FUNCTION_BLOCK TcoTixonVibro_v_1_x_x EXTENDS TcoCore.TcoComponent
VAR_INPUT
    inControllerInAuto : BOOL;
    inNotEmptyFeeder : BOOL;
    inSeparatorHomePos : BOOL;
    inFillingSensor : BOOL;
    inSeparatorPresent : BOOL;
    inComponentOutOfBox : BOOL;
    inSeparatorWorkPos : BOOL;
END_VAR
VAR_OUTPUT
    outFeedingA : BOOL;
    outSepareComponent : BOOL;
    outBlowValveA : BOOL;
    outRedLed : BOOL;
    outGreenLed : BOOL;
    outHopper : BOOL;
    outShotComponent : BOOL;
END_VAR
VAR
    {attribute addProperty Name "<#Status#>"}
    {attribute clr [ReadOnly()]}
    _status : TcoTixonVibro_Status_v_1_x_x;
    {attribute addProperty Name "<#Control#>"}
    _control : TcoTixonVibro_Control_v_1_x_x;
    {attribute addProperty Name "<#Config#>"}
    _config : TcoTixonVibro_Config_v_1_x_x;
    _someTaskIsActive : BOOL;
    {attribute 'hide'}
    _blink : TcoUtilities.TcoBlinker(THIS^);
    _runAutomatic : BOOL;
    _hasError : BOOL;
END_VAR
VAR
    {attribute addProperty Name "<#Separator task#>"}
    _separatorTask : TcoTixonVibroSeparatorTask(THIS^);
    {attribute addProperty Name "<#Buffer task#>"}
    _bufferTask : TcoTixonBufferTask(THIS^);
    {attribute addProperty Name "<#Hopper task#>"}
    _hopperTask : TcoTixonHopperTask(THIS^);
    {attribute addProperty Name "<#Restore#>"}
    _restoreTask : TcoCore.TcoTask(THIS^);
END_VAR
VAR
    {attribute 'hide'}
    _sb : TcoCore.StringBuilder;
END_VAR

_blink(inOnTime := _config.BlinkTime, inOffTime := _config.BlinkTime);
UpdateStatus();
_separatorTask.Enabled := TRUE;
_separatorTask.ErrorTime := _config.ErrorTimeSeparator;
_separatorTask(inoConfig := _config, inoControl := _control, inoStatus := _status);
_bufferTask.Enabled := TRUE;
_bufferTask.ErrorTime := _config.ErrorTimeBuffer;
_bufferTask(inoConfig := _config, inoControl := _control, inoStatus := _status);
_hopperTask.ErrorTime := _config.ErrorTimeHopper;
_hopperTask.Enabled := _config.HopperActive;
_hopperTask(inoConfig := _config, inoControl := _control, inoStatus := _status);
//*************RESTORE********************
_restoreTask.Enabled := TRUE;

IF _restoreTask.Execute() THEN
    Restore();
    _restoreTask.DoneWhen(TRUE);
END_IF
//****************************************
UpdateControl();

METHOD PUBLIC BufferFeed : TcoCore.ITcoTaskStatus
BufferFeed := _bufferTask.Invoke();
_bufferTask.AutoRestore := false;
END_METHOD

PROPERTY PUBLIC BufferTask : REFERENCE TO TcoTixonBufferTask
GET
BufferTask ref= _bufferTask;
END_GET
END_PROPERTY

(*~
    <docu>
        <summary>
            Gets the configuration of the Tixon Vibro.
        </summary>
    </docu>
~*)
PROPERTY Config : REFERENCE TO TcoTixonVibro_Config_v_1_x_x
GET
Config REF= _config;
END_GET
END_PROPERTY

METHOD PUBLIC CyclicBufferFeed : TcoCore.ITcoTaskStatus
CyclicBufferFeed := _bufferTask.Invoke();
_bufferTask.AutoRestore := true;
END_METHOD

METHOD PUBLIC CyclicHopperFeed : TcoCore.ITcoTaskStatus
CyclicHopperFeed := _hopperTask.Invoke();
_hopperTask.AutoRestore := TRUE;
END_METHOD

METHOD PUBLIC CyclicSepare : TcoCore.ITcoTaskStatus
CyclicSepare := _separatorTask.Invoke();
_separatorTask.AutoRestore := true;
END_METHOD

METHOD PUBLIC DefaultSignalisation
VAR_INPUT
END_VAR
// led signalisation
_hasError := _separatorTask.Error OR _bufferTask.Error OR _hopperTask.Error;
_control.GreenLed := FALSE;
_control.RedLed := FALSE;

IF NOT _status.ControllerInAuto THEN
    _control.GreenLed := TRUE;
    _control.RedLed := TRUE;
ELSIF _hasError AND _blink.IsOn AND _status.ControllerInAuto THEN
    _control.RedLed := TRUE;
ELSIF _status.ControllerInAuto AND NOT _hasError AND _status.NotEmptyFeeder THEN
    _control.GreenLed := TRUE;
ELSIF _blink.IsOn AND _status.ControllerInAuto AND NOT _status.NotEmptyFeeder THEN
    _control.GreenLed := TRUE;
    _control.RedLed := TRUE;
END_IF
END_METHOD

METHOD PUBLIC HopperFeed : TcoCore.ITcoTaskStatus
HopperFeed := _hopperTask.Invoke();
_hopperTask.AutoRestore := false;
END_METHOD

PROPERTY PUBLIC HopperTask : reference TO TcoTixonHopperTask
GET
HopperTask ref= _hopperTask;
END_GET
END_PROPERTY

METHOD PUBLIC Push
VAR_INPUT
    inReqOn : BOOL;
END_VAR
_control.ShotComponent := inReqOn;
END_METHOD

(*~
    <docu>
        <summary>
            Restores this instance to the Ready state. Can be called explicitly or from within one of the restore mechanisms.
        </summary>
    </docu>
~*)
METHOD Restore : ITcoRestorable
RestoreTasks();
_control.BlowAValve := FALSE;
_control.FeedingA := FALSE;
_control.GreenLed := FALSE;
_control.RedLed := FALSE;
_control.SepareComponent := FALSE;
_control.ShotComponent := FALSE;
_control.Hooper := FALSE;
END_METHOD

METHOD INTERNAL RestoreTasks
_separatorTask.Restore();
_bufferTask.Restore();
_hopperTask.Restore();
END_METHOD

PROPERTY PUBLIC SeparatorTask : REFERENCE TO TcoTixonVibroSeparatorTask
GET
SeparatorTask ref= _separatorTask;
END_GET
END_PROPERTY

METHOD PUBLIC Separe : TcoCore.ITcoTaskStatus
Separe := _separatorTask.Invoke();
_separatorTask.AutoRestore := false;
END_METHOD

(*~
    <docu>
        <summary>
            Custom service (manual, maintenance) logic.
            This method must be implemented in derived class.
        </summary>
    </docu>
~*)
METHOD PROTECTED ServiceMode
END_METHOD

(*~
    <docu>
        <summary>
            Gets the status of the Tixon Vibro.
        </summary>
    </docu>
~*)
PROPERTY Status : REFERENCE TO TcoTixonVibro_Status_v_1_x_x
GET
Status REF= _status;
END_GET
END_PROPERTY

METHOD INTERNAL UpdateControl
VAR_INPUT
END_VAR
VAR
    index : INT;
END_VAR
outBlowValveA := _control.BlowAValve;
outFeedingA := _control.FeedingA;
outGreenLed := _control.GreenLed;
outRedLed := _control.RedLed;
outSepareComponent := _control.SepareComponent;
outShotComponent := _control.ShotComponent;
outHopper := _control.Hooper;
END_METHOD

METHOD INTERNAL UpdateStatus
VAR
END_VAR
_status.ComponentOutOfBox := inComponentOutOfBox;
_status.NotEmptyFeeder := inNotEmptyFeeder;
_status.FillingSensor := inFillingSensor;
_status.SeparatorHomePos := inSeparatorHomePos;
_status.SeparatorPresent := inSeparatorPresent;
_status.ControllerInAuto := inControllerInAuto;
_status.SeparatorWorkPos := inSeparatorWorkPos;
END_METHOD

END_FUNCTION_BLOCK

(* stored: Version 1.1.0.1, ProductVersion 3.1.4024.12
   POU TcoTixonVibro_v_1_x_x: Id {ef7e1a36-bdd5-06f3-2c86-7faf9d79ac2a}, SpecialFunc None
   Folder Operations: Id {dcfc56ef-b55c-06df-2430-f7dd1bd8c181}
   Folder Loop: Id {e17e7df9-8969-0354-1a79-3426342e693b}
   Folder Single: Id {dea1b71d-4204-0383-06d1-cc70ee27325d}
   Folder Task: Id {cb53b1a0-e58a-0097-1ad4-6d3d1414fabb}
   Method BufferFeed: Id {523e43d6-1bff-0ba1-34f7-38e8a7e28910}
   Property BufferTask: Id {6e3d1d3e-cd2b-0993-1f43-2d3bfaa7e320}
   Get Get: Id {c9298ad1-f7e2-0d65-2a3f-612351825685}
   Property Config: Id {f965d48e-b1c0-0055-2c7f-992887c08b4d}
   Get Get: Id {542b70eb-e6e3-032d-34b4-c7e888300a8b}
   Method CyclicBufferFeed: Id {f210448c-2fdd-0675-1acc-9cffd3d6c8c9}
   Method CyclicHopperFeed: Id {fc238180-fc20-0806-2762-83b25f612f90}
   Method CyclicSepare: Id {1dee92ea-80a4-01a4-3ce1-31280b8d546f}
   Method DefaultSignalisation: Id {c1b303a8-c50a-041f-2d52-a1fdae8aaed4}
   Method HopperFeed: Id {fbbf6aa4-5fdc-0146-0cd5-3e55b7ce0886}
   Property HopperTask: Id {4e88dc4b-f856-0175-1dc3-f1259469d210}
   Get Get: Id {1d115ad8-d104-0fc9-349b-e1adfe3c7c91}
   Method Push: Id {440f6881-cda9-0a40-2000-bd324270cce8}
   Method Restore: Id {b77c9cd5-75e1-059b-1d7d-ad2222006348}
   Method RestoreTasks: Id {6b5ae874-ab97-0567-19e8-4381140720a2}
   Property SeparatorTask: Id {5bb208cb-75e5-0a0c-2de4-0a97eb7537fd}
   Get Get: Id {bc50ad8a-a15d-00e3-23b6-b145b78d5122}
   Method Separe: Id {22addfa8-500f-0608-2ff3-619118af22b8}
   Method ServiceMode: Id {1680ba29-57a9-0ff3-2da1-54e60a3f2225}
   Property Status: Id {9caf956e-bed1-0082-00a2-de7cf3bc52b1}
   Get Get: Id {11dc26cb-49d1-0876-1ff7-2cce3331d67e}
   Method UpdateControl: Id {9d5e82ce-ac09-0f4a-3766-e32a9b69c1cd}
   Method UpdateStatus: Id {47aa9dae-4833-007a-38a6-dc199b41f6e3} *)
